Omron Sysmac Studio project CIPSafety_TURCK (Sysmac Studio 1.54.0.64019, StandardProject)

# Controller new_Controller_0: NX102-1220 version 1.48
Units and slaves: Unit 2 : NX-ILM400 (N2)
Task PrimaryTask (priority 4, period or condition 2000): Program0

TYPE TURCK_CIP : STRUCT
    FieldbusBits : ARRAY[0..15] of bool;
    StationStatus : TURCK_CIPSafety_StationStatusWord;
    SafetyStatus : TURCK_CIPSafety_Status;
    SafetyCx : ARRAY[0..7] OF TURCK_CIPSafety_CxStatus;
    ModuleStatus : TURCK_CIPSafety_ModuleStatus;
END_STRUCT END_TYPE
TYPE TURCK_CIPSafety_StationStatusWord : STRUCT
    ModuleDiagnosticsAvailable : BOOL;
    StationConfiguredChanged : BOOL;
    OverCurrentIsys : BOOL;
    OverVoltageV2 : BOOL;
    UnderVoltageV2 : BOOL;
    OverVoltageV1 : BOOL;
    UnderVoltageV1 : BOOL;
    ModuleBusCoumLost : BOOL;
    ModuleBusError : BOOL;
    ForceModeEnabled : BOOL;
END_STRUCT END_TYPE
TYPE TURCK_CIPSafety_Status : STRUCT
    ProtectiveMode : BOOL;
    ConfigurationMode : BOOL;
    UnKnownMode : BOOL;
    NoMemoryStick : BOOL;
    NoConfigurationAvailable : BOOL;
    ConfigurationMismatch : BOOL;
    CommunicationLoss : BOOL;
    FateError : BOOL;
END_STRUCT END_TYPE
TYPE TURCK_CIPSafety_CxStatus : STRUCT
    Normal : BOOL;
    WaitForInput : BOOL;
    TestInput : BOOL;
    InputError : BOOL;
    CrossCircuitCh0 : BOOL;
    CrossCircuitCh1 : BOOL;
    OutputOverload : BOOL;
END_STRUCT END_TYPE
TYPE TURCK_CIPSafety_ModuleStatus : STRUCT
    IOAssistantForceMode : BOOL;
    UnderVoltage1 : BOOL;
    UnderVoltage2 : BOOL;
    ModuleDiagnosticsAvailable : BOOL;
    InternalError : BOOL;
END_STRUCT END_TYPE
TYPE Byte2Bool : UNION
    BoolData : ARRAY[0..7] OF bool;
    ByteData : BYTE;
END_UNION END_TYPE
TYPE TURCK_CIP_Outputs : STRUCT
    TURCK_CIP_Outputs_SafetyStatus : BOOL;
    TURCK_CIP_Outputs_FieldBits : ARRAY[0..15] of bool;
END_STRUCT END_TYPE

VAR_GLOBAL
    Turck_Module1 : TURCK_CIP;
    dataFromTurck : ARRAY[0..19] OF Byte;  (* network input *)
    dataFromPilz : ARRAY[0..31] OF byte;  (* network input *)
    dataToTurck : ARRAY[0..5] OF byte;  (* network output *)
    dataToPilz : ARRAY[0..31] OF byte;  (* network output *)
END_VAR

(* Program Program0: safety or other program stored in binary form, left out *)

PROGRAM Program0
VAR
    FB_TURCKCIPSafety1 : FB_TURCKCIPSafety;
    ESTOPStatus : BOOL;
    FieldbusBitON : BOOL;
    FieldbusBitOFF : BOOL;
END_VAR
VAR_EXTERNAL
    dataFromTurck : ARRAY[0..19] OF Byte;
    Turck_Module1 : TURCK_CIP;
    dataToTurck : ARRAY[0..5] OF byte;
END_VAR

(* Section Section0: ladder, written here as Structured Text *)

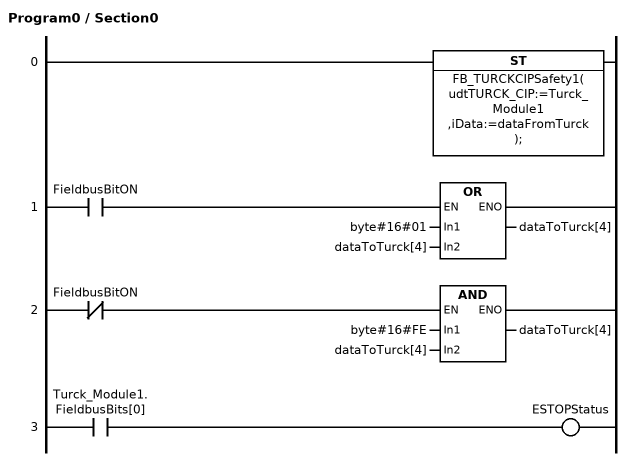
(* Rung 0 *)
FB_TURCKCIPSafety1(
	udtTURCK_CIP:=Turck_Module1
	,iData:=dataFromTurck
	);
(* Rung 1 *)
IF FieldbusBitON THEN dataToTurck[4] := byte#16#01 OR dataToTurck[4]; END_IF;
(* Rung 2 *)
IF NOT FieldbusBitON THEN dataToTurck[4] := byte#16#FE AND dataToTurck[4]; END_IF;
(* Rung 3 *)
ESTOPStatus := Turck_Module1.FieldbusBits[0];
END_PROGRAM

FUNCTION FC_GetCxStatus : BOOL
VAR
    uByte2Bool : Byte2Bool;
END_VAR
VAR_INPUT
    iByte1 : BYTE;
END_VAR
VAR_IN_OUT
    udtCxStatus : TURCK_CIPSafety_CxStatus;
END_VAR
uByte2Bool.ByteData:=iByte1;

udtCxStatus.Normal:=uByte2Bool.BoolData[0];
udtCxStatus.WaitForInput:=uByte2Bool.BoolData[1];
udtCxStatus.TestInput:=uByte2Bool.BoolData[2];
udtCxStatus.InputError:=uByte2Bool.BoolData[3];
udtCxStatus.CrossCircuitCh0:=uByte2Bool.BoolData[4];
udtCxStatus.CrossCircuitCh1:=uByte2Bool.BoolData[5];
udtCxStatus.OutputOverload:=uByte2Bool.BoolData[7];
END_FUNCTION

FUNCTION_BLOCK FB_TURCKCIPSafety
VAR
    uByte2Bool : Byte2Bool;
END_VAR
VAR_IN_OUT
    udtTURCK_CIP : TURCK_CIP;
END_VAR
VAR_INPUT
    iData : ARRAY[0..19] OF byte;
END_VAR
uByte2Bool.ByteData:=iData[0];

//Station Status word
	uByte2Bool.ByteData:=iData[0];//word0
	udtTURCK_CIP.StationStatus.ModuleDiagnosticsAvailable:=uByte2Bool.BoolData[0];
	udtTURCK_CIP.StationStatus.StationConfiguredChanged:=uByte2Bool.BoolData[3];
	udtTURCK_CIP.StationStatus.OverCurrentIsys:=uByte2Bool.BoolData[5];
	udtTURCK_CIP.StationStatus.OverVoltageV2:=uByte2Bool.BoolData[6];
	udtTURCK_CIP.StationStatus.UnderVoltageV2:=uByte2Bool.BoolData[7];
	
	uByte2Bool.ByteData:=iData[1];//word0
	udtTURCK_CIP.StationStatus.OverVoltageV1:=uByte2Bool.BoolData[0];	//8
	udtTURCK_CIP.StationStatus.UnderVoltageV2:=uByte2Bool.BoolData[1];	//9
	udtTURCK_CIP.StationStatus.ModuleBusCoumLost:=uByte2Bool.BoolData[2]; //10
	udtTURCK_CIP.StationStatus.ModuleBusError:=uByte2Bool.BoolData[3]; //11
	udtTURCK_CIP.StationStatus.ForceModeEnabled:=uByte2Bool.BoolData[6]; //14

//Safety Status
	uByte2Bool.ByteData:=iData[2];//word1 byte2,3
	udtTURCK_CIP.SafetyStatus.ProtectiveMode:=uByte2Bool.BoolData[0];
	udtTURCK_CIP.SafetyStatus.ConfigurationMode:=uByte2Bool.BoolData[1];
	udtTURCK_CIP.SafetyStatus.UnKnownMode:=uByte2Bool.BoolData[2];
	
	uByte2Bool.ByteData:=iData[4];//word2 byte4,5
	
	uByte2Bool.ByteData:=iData[6];//word3 byte6,7
	udtTURCK_CIP.SafetyStatus.NoMemoryStick:=uByte2Bool.BoolData[0];
	udtTURCK_CIP.SafetyStatus.NoConfigurationAvailable:=uByte2Bool.BoolData[1];
	udtTURCK_CIP.SafetyStatus.ConfigurationMismatch:=uByte2Bool.BoolData[2];
	udtTURCK_CIP.SafetyStatus.CommunicationLoss:=uByte2Bool.BoolData[4];
	udtTURCK_CIP.SafetyStatus.FateError:=uByte2Bool.BoolData[7];
	
	uByte2Bool.ByteData:=iData[8];//word4 byte8
	FC_GetCxStatus(
		EN:=TRUE
		,iByte1:=iData[8]
		,udtCxStatus:=udtTURCK_CIP.SafetyCx[0]
		);
	
	uByte2Bool.ByteData:=iData[9];//word4 byte9
	FC_GetCxStatus(
		EN:=TRUE
		,iByte1:=iData[9]
		,udtCxStatus:=udtTURCK_CIP.SafetyCx[1]
		);

	uByte2Bool.ByteData:=iData[10];//word5 byte10
	FC_GetCxStatus(
		EN:=TRUE
		,iByte1:=iData[10]
		,udtCxStatus:=udtTURCK_CIP.SafetyCx[2]
		);
	
	uByte2Bool.ByteData:=iData[11];//word5 byte11
	FC_GetCxStatus(
		EN:=TRUE
		,iByte1:=iData[11]
		,udtCxStatus:=udtTURCK_CIP.SafetyCx[3]
		);

	uByte2Bool.ByteData:=iData[12];//word6 byte12
	FC_GetCxStatus(
		EN:=TRUE
		,iByte1:=iData[11]
		,udtCxStatus:=udtTURCK_CIP.SafetyCx[4]
		);
	uByte2Bool.ByteData:=iData[13];//word6 byte13
	FC_GetCxStatus(
		EN:=TRUE
		,iByte1:=iData[11]
		,udtCxStatus:=udtTURCK_CIP.SafetyCx[5]
		);
	
	uByte2Bool.ByteData:=iData[14];//word7 byte14
	FC_GetCxStatus(
		EN:=TRUE
		,iByte1:=iData[11]
		,udtCxStatus:=udtTURCK_CIP.SafetyCx[6]
		);
	
	uByte2Bool.ByteData:=iData[15];//word7 byte15
	FC_GetCxStatus(
		EN:=TRUE
		,iByte1:=iData[11]
		,udtCxStatus:=udtTURCK_CIP.SafetyCx[7]
		);
	
	uByte2Bool.ByteData:=iData[16];//word8 Byte16
	udtTURCK_CIP.FieldbusBits[0]:=uByte2Bool.BoolData[0];
	udtTURCK_CIP.FieldbusBits[1]:=uByte2Bool.BoolData[1];
	udtTURCK_CIP.FieldbusBits[2]:=uByte2Bool.BoolData[2];
	udtTURCK_CIP.FieldbusBits[3]:=uByte2Bool.BoolData[3];
	udtTURCK_CIP.FieldbusBits[4]:=uByte2Bool.BoolData[4];
	udtTURCK_CIP.FieldbusBits[5]:=uByte2Bool.BoolData[5];
	udtTURCK_CIP.FieldbusBits[6]:=uByte2Bool.BoolData[6];
	udtTURCK_CIP.FieldbusBits[7]:=uByte2Bool.BoolData[7];

	uByte2Bool.ByteData:=iData[17];//word8 Byte17
	udtTURCK_CIP.FieldbusBits[8]:=uByte2Bool.BoolData[0];
	udtTURCK_CIP.FieldbusBits[9]:=uByte2Bool.BoolData[1];
	udtTURCK_CIP.FieldbusBits[10]:=uByte2Bool.BoolData[2];
	udtTURCK_CIP.FieldbusBits[11]:=uByte2Bool.BoolData[3];
	udtTURCK_CIP.FieldbusBits[12]:=uByte2Bool.BoolData[4];
	udtTURCK_CIP.FieldbusBits[13]:=uByte2Bool.BoolData[5];
	udtTURCK_CIP.FieldbusBits[14]:=uByte2Bool.BoolData[6];
	udtTURCK_CIP.FieldbusBits[15]:=uByte2Bool.BoolData[7];
	
	uByte2Bool.ByteData:=iData[18];//word9 Byte18
	udtTURCK_CIP.ModuleStatus.ModuleDiagnosticsAvailable:=uByte2Bool.BoolData[0];
	udtTURCK_CIP.ModuleStatus.UnderVoltage2:=uByte2Bool.BoolData[7];
	
	uByte2Bool.ByteData:=iData[18];//word9 Byte19
	udtTURCK_CIP.ModuleStatus.UnderVoltage1:=uByte2Bool.BoolData[1];
	udtTURCK_CIP.ModuleStatus.InternalError:=uByte2Bool.BoolData[2];
	udtTURCK_CIP.ModuleStatus.IOAssistantForceMode:=uByte2Bool.BoolData[6];
	
END_FUNCTION_BLOCK